SUBAPPLICATION Uebung_002b3 (* DigitalInput_I1/_I2/_I3 auf DigitalOutput_Q1; ohne MOVE *)
  (* Standard: 61499-2; Description: Copyright (c) 2023 Meisterschulen am Ostbahnhof This program and the accompanying materials are made available under the terms of the Eclipse Public License 2.0 which is available at https://www.eclipse.org/legal/epl-2.0/ SPDX-License-Identifier: EPL-2.0 *)
  (* Version 1.0, 2023-10-23, Franz Höpfinger, Meisterschulen am Ostbahnhof, initial API and implementation and/or initial documentation *)
  PACKAGE Uebungen;
  IMPORT logiBUS::io::DI::logiBUS_DI::Input_I1;
  IMPORT logiBUS::io::DI::logiBUS_DI::Input_I2;
  IMPORT logiBUS::io::DI::logiBUS_DI::Input_I3;
  IMPORT logiBUS::io::DQ::logiBUS_DO::Output_Q1;
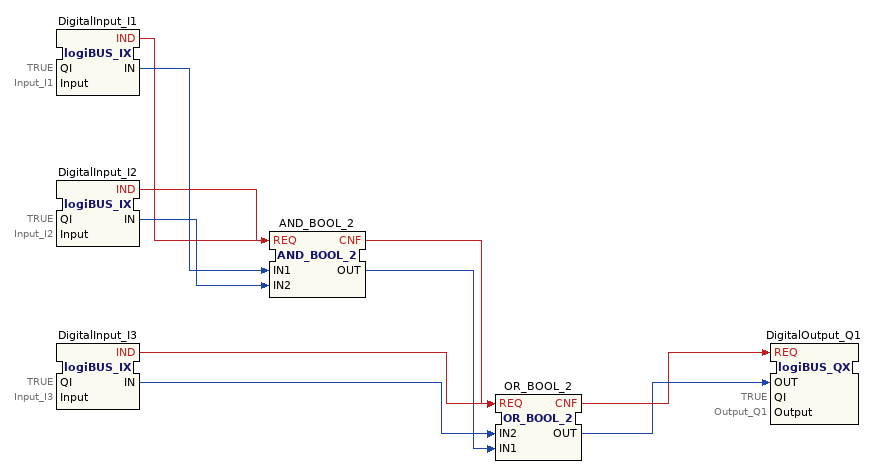
  (* kein F_MOVE mehr nötig. *)
  FBS
    DigitalOutput_Q1 : logiBUS::io::DQ::logiBUS_QX(QI := TRUE, Output := Output_Q1);
    DigitalInput_I1 : logiBUS::io::DI::logiBUS_IX(QI := TRUE, Input := Input_I1);
    DigitalInput_I2 : logiBUS::io::DI::logiBUS_IX(QI := TRUE, Input := Input_I2);
    AND_BOOL_2 : iec61131::booleanOperators::AND_BOOL_2;
    DigitalInput_I3 : logiBUS::io::DI::logiBUS_IX(QI := TRUE, Input := Input_I3);
    OR_BOOL_2 : iec61131::booleanOperators::OR_BOOL_2;
  END_FBS
  EVENT_CONNECTIONS
    DigitalInput_I1.IND TO AND_BOOL_2.REQ;
    DigitalInput_I2.IND TO AND_BOOL_2.REQ;
    OR_BOOL_2.CNF TO DigitalOutput_Q1.REQ;
    DigitalInput_I3.IND TO OR_BOOL_2.REQ;
    AND_BOOL_2.CNF TO OR_BOOL_2.REQ;
  END_CONNECTIONS
  DATA_CONNECTIONS
    DigitalInput_I1.IN TO AND_BOOL_2.IN1;
    DigitalInput_I2.IN TO AND_BOOL_2.IN2;
    DigitalInput_I3.IN TO OR_BOOL_2.IN2;
    OR_BOOL_2.OUT TO DigitalOutput_Q1.OUT;
    AND_BOOL_2.OUT TO OR_BOOL_2.IN1;
  END_CONNECTIONS
END_SUBAPPLICATION
